PROGRAM MAIN
VAR
	TheThing	: FB_TheThing;
	OtherThing	: FB_OtherThing;
END_VAR

thething();
IF theThing.prepare_to_do_the_thing() THEN
	theThing.do_the_thing();
END_IF

END_PROGRAM

(* stored: Version 1.1.0.1, ProductVersion 3.1.4024.0
   POU MAIN: Id {3163ddc5-cc52-4a07-903d-877f782f00da}, SpecialFunc None *)
